(* PLC project Tc2_Utilities.FB_EnumFindFileEntry Demo, tc3-libraries-kb TwinCAT 3.1 *)
(* stored: creationDateTime 2026-05-11T13:00:00, modificationDateTime 2026-05-11T13:00:00 *)

PROGRAM P_Demo_FB_EnumFindFileEntry
  VAR
    fbFB_EnumFindFileEntry : FB_EnumFindFileEntry;  (* FB_EnumFindFileEntry 实例 *)
    sNetID : T_AmsNetID := '';
    sPathName : T_MaxString := '';
    eCmd : E_EnumCmdType := eEnumCmd_First;
    bExecute : BOOL := FALSE;
    tTimeout : TIME := DEFAULT_ADS_TIMEOUT;
    bBusy : BOOL;
    bError : BOOL;
    nErrId : UDINT;
    bEOE : BOOL;
    stFindFile : ST_FindFileEntry;
  END_VAR

// =============================================================================
// 场景：FB_EnumFindFileEntry 的最小可编译演示——所有 VAR_INPUT 均以 doc/PDF 中真实引脚名调用。
//       业务侧请在线 monitor / 在线写值触发对应输入，看输出端 monitor 结果。
//
// 价值：保证示例 ST 代码所有引脚名与 FB_EnumFindFileEntry 的 VAR_INPUT/VAR_OUTPUT 一致，
//       Import PLCopenXML → 编译 → 登录 流程能跑通，作为 hand-curated 例程
//       的脚手架。
//
// 验证步骤：
//   1. 引用 Tc2_Utilities（及其依赖 Tc2_System）
//   2. 右键 PLC 项目 → Import PLCopenXML → 选本文件 → OK → 编译、登录
//   3. 在线对 VAR_INPUT 写入合适触发值（典型 bExecute / RUN / START 上升沿）
//   4. 在线 monitor VAR_OUTPUT 观察 FB 反应
// =============================================================================

fbFB_EnumFindFileEntry(
    sNetID := sNetID,
    sPathName := sPathName,
    eCmd := eCmd,
    bExecute := bExecute,
    tTimeout := tTimeout,
    bBusy => bBusy,
    bError => bError,
    nErrId => nErrId,
    bEOE => bEOE,
    stFindFile => stFindFile
);
END_PROGRAM
